Staubli VAL3: modIMM.pjx

--- modIMM.pjx ---
Parameters version=s7.2 stackSize=5000 millimeterUnit=true
Program file=_StartMachine.pgx
Program file=_WaitAuto.pgx
Program file=_WaitEnd.pgx
Program file=_WaitPart.pgx
Program file=_WaitPartDyn.pgx
Program file=BtRobotOff.pgx
Program file=checkMotStack.pgx
Program file=childAction.pgx
Program file=getSetting.pgx
Program file=IMMTiming.pgx
Program file=init.pgx
Program file=loadLibraries.pgx
Program file=primeAreaTest.pgx
Program file=primeMotStack.pgx
Program file=registerSetting.pgx
Program file=retrieveViews.pgx
Program file=runHigh.pgx
Program file=runLow.pgx
Program file=secuTask1.pgx
Program file=secuTask2.pgx
Program file=setDryRunSig.pgx
Program file=setSetting.pgx
Program file=slot.pgx
Program file=start.pgx
Program file=startAreaTest.pgx
Program file=stop.pgx
Program file=stopAreaTest.pgx
Program file=taskPartMade.pgx
Program file=updateView.pgx
Program file=WaitPart.pgx
Data file=modIMM.dtx
Library alias=io path=Disk://io/io.pjx
Library alias=SYS path=Disk://io_System/io_System.pjx
Library alias=scr path=Disk://Plastic/coreModules/modScreen/modScreen.pjx
Library alias=str path=Disk://Libraries/stringHandling/stringHandling.pjx
Library alias=lang path=Disk://Plastic/i18n/i18n.pjx
Library alias=debug path=Disk://Libraries/debug/debug.pjx
Library alias=data path=Disk://zData/zData.pjx
Library alias=status path=Disk://Plastic/coreModules/modStatusModel/modStatusModel.pjx
Library alias=EV path=Disk://Plastic/Consts/EVENT/EVENT.pjx
Library alias=sig path=Disk://Plastic/coreModules/modSignalSlot/modSignalSlot.pjx
Library alias=STATE path=Disk://Plastic/Consts/STATE/STATE.pjx
Library alias=views path=Disk://Plastic/coreModules/viewContainer/viewContainer.pjx
Library alias=jt path=Disk://Libraries/jointFunctions/jointFunctions.pjx
Type name=event path=Disk://Plastic/Types/event/event.pjx
Type name=settingType path=Disk://Plastic/Types/setting/setting.pjx
Type name=viewType path=Disk://Plastic/Types/view/view.pjx
Type name=childNodeType path=Disk://Plastic/Types/childNode/childNode.pjx
Type name=nodeType path=Disk://Plastic/Types/node/node.pjx

--- modIMM.dtx ---
num nCaseBtRobOff
num nStateRstPart[4]
num nStatePartMade
num reactionTime
num pointer
num timings[40]
public num nCloseDelayTime
num mouldTimer
bool bRobotOffAllow
bool bState
num tmMotionStack
num WAR_MOTIONSTACK = 1
bool bDisplayed
bool bSuspendForTest
num WAIT_MOULD_FREE
num nAreaTestState
num nMouldAreaZone
num WAIT_MOULD_OPEN
num WAIT_ROB_ENABLE
num WAIT_IMM_AUTO
num WAIT_PARTMADE
public string name = "IMM"
num moduleIndex
bool bAtWaitPosition
string IMM_IO_PTH
num nImmType
bool bRobotOff
num AREA_TEST_FAIL
num nMouldAreaDist
num HOME_IN_MOULD
num ARM_IN_MOULD_NO
num ARM_IN_MOULD_ST

--- start.pgx ---
public program start()
begin
  // set nCaseBtRobOff to 1 instead of 0 in order to initialize the robot off function properly
  // If nCaseBtRobOff is 0 at start up it may happen that SYS:doRobotOff["+toString("",moduleIndex)+"] is on although btRobotOff assumes that
  // SYS:doRobotOff["+toString("",moduleIndex)+"] is off.

  call debug:setVerbosity(libPath(),debug:LEV_INFO)
  call loadLibraries()
  // call setDryRunSig(data:setDryRun)
  call sig:connect(EV:DRY_RUN,libPath())
  call sig:connect(EV:FATAL_ERROR,libPath())
  call sig:connect(EV:START_COMPLETE,libPath())
  call status:registerStatus(libPath(),status:CL_STATUS,"Wait for mould free condition","SYS:doMouldFree["+toString("",moduleIndex)+"]==true","SYS:doMouldFree["+toString("",moduleIndex)+"]==false",false,WAIT_MOULD_FREE,false)
  call status:registerStatus(libPath(),status:CL_STATUS,"Wait for mould open","SYS:diMouldOpen["+toString("",moduleIndex)+"]==true","SYS:diMouldOpen["+toString("",moduleIndex)+"]==false",false,WAIT_MOULD_OPEN,false)
  call status:registerStatus(libPath(),status:CL_STATUS,"Wait for robot enabled","SYS:doRobotOff["+toString("",moduleIndex)+"]==false","SYS:doRobotOff["+toString("",moduleIndex)+"]==true",false,WAIT_ROB_ENABLE,false)
  call status:registerStatus(libPath(),status:CL_STATUS,"Wait for IMM in auto mode","SYS:diMachineInAuto["+toString("",moduleIndex)+"]==true","SYS:diMachineInAuto["+toString("",moduleIndex)+"]==false",false,WAIT_ROB_ENABLE,false)
  call status:registerStatus(libPath(),status:CL_STATUS,"Wait for part produced","SYS:bPartMade["+toString("",moduleIndex)+"]==true","SYS:bPartMade["+toString("",moduleIndex)+"]==false",false,WAIT_PARTMADE,false)
  call status:registerStatus(libPath(),status:CL_ERROR,"Mould area test failed. Robot was not programmed to enter mould","","",true,AREA_TEST_FAIL,true)
  call status:registerStatus(libPath(),status:CL_ERROR,"Home position is defined in mould area","","",true,HOME_IN_MOULD,true)
  call status:registerStatus(libPath(),status:CL_ERROR,"Arm in mould while mould is not open","","",true,ARM_IN_MOULD_NO,true)
  call status:registerStatus(libPath(),status:CL_ERROR,"Arm in mould while 'Enable Closure' signal is set","","",true,ARM_IN_MOULD_ST,true)
end

--- _StartMachine.pgx ---
public program _StartMachine()
// Start machine cycle
  local bool bAreaTest
  local num nOldSpeedScale
  local bool bTestRun
  local string txt
  local num time
  local string sValue
begin
  //
  // add list of pending status messages
  //!i18n 16 -> "Wait for Mould Free Condition"

  call status:setEnabled(WAIT_MOULD_FREE,true)
  //!change 23.05.06, vdg: reduce speed in test mode when approaching the mould area boundary
  // from inside towards outside
  //!change 08.09.06, vdg: store data:setTestRun in a local variable
  bTestRun=data:setTestRun
  // prime the motion stack monitor which checks if the arm is actually
  // programmed to leave the mould when StartMachine() is called
  call primeMotStack()
  if bTestRun
    //wait(secu:nSafeZoneDist[0]<300)
    nOldSpeedScale=getMonitorSpeed()
    //!fix 09.06.06, vdg: set speed to the lower speed setting (current speedScale() or dry run speed)
    ///TODO
    //$setSpeed(min(speedScale(),10))
    //call setSpeed(min(getMonitorSpeed(),10))
    //wait(secu:nSafeZoneDist[0]<50)
    //$setSpeed(1)
    ///TODO
    //call setSpeed(1)
  endIf
  // WAIT GRIPPER OUT OF MOULD AREA ==================================================================================
  // record the safety distance of the robot

  time=clock()
  //requiredTime=0.2
  //currentTime=0
  // if (speedScale()>99) and (workingMode()==4) and (SYS:diMachineInAuto[moduleIndex]==true) and !bTestRun
  if (getMonitorSpeed()>99) and (workingMode()==4) and !bTestRun
    do
      // Check if there are still motions in the stack.
      // If it is empty, it means the robot never leaves the mould area before
      // StartMachine() is called.
      call checkMotStack()
    until (SYS:doMouldFree[moduleIndex]==true)
  else
    do
      // Check if there are still motions in the stack.
      // If it is empty, it means the robot never leaves the mould area before
      // StartMachine() is called.
      call checkMotStack()
    until (SYS:doMouldFree[moduleIndex]==true)
  endIf
  //
  call status:setEnabled(WAIT_MOULD_FREE,false)
  //
  //!change 18.05.06, vdg: check if doMouldFree has toggled
  call stopAreaTest(bAreaTest)
  // START MACHINE CYCLE =============================================================================================
  //!change 16.02.06, vdg: Allow to start IMM in endIf cycle mode SYS:bStartInEndCycl is set
  if (!SYS:CE_Requested or SYS:bStartInEndCycl) and !SYS:bPartMade[moduleIndex] and bAreaTest
    //!change 18.05.06, vdg: Stop robot at point where machine is being started
    //  and ask the user if it is safe to start the IMM
    if bTestRun
      bSuspendForTest=true
      // reset original speedScale only if speed was not modified by user meanwhile
      // wait for settled arm
      watch(isSettled(),3)
      // reset old speed setting if it wasn't changed by the user
      if getMonitorSpeed()==1
        ///TODO
        //$setSpeed(nOldSpeedScale)
        //call setSpeed(nOldSpeedScale)
      endIf
      //sValue=toString("4.0",secu:nSafeZoneDist[0])
      call str:printf((("Robot stopped approx. at point where IMM cycle is being started (Overshoot: %1mm). Press START to continue!")),sValue,txt)
      ///TODO
      //call ui:popUpCond(txt,"SYS:bBtStart==true",false)
      bSuspendForTest=true
      wait(bSuspendForTest==false)
    endIf
    //!change 08.06.06, vdg: Start IMM only if dry run mode is not active
    if !bTestRun
      SYS:doStartMachine[moduleIndex]=true
    endIf
    //call stat:stopTakeTime()
    //call stat:stopCycleTime()
    //call stat:startCycleTime()
    //call stat:startRobotTime()
  endIf
  //
end

--- _WaitPartDyn.pgx ---
public program _WaitPartDyn()
// Wait part made in machine and mould fully open
begin
  //!brief
  // Wait for a part being made and conditions for the robot to enter mold.
  //
  call WaitPart(true)
end

--- checkMotStack.pgx ---
program checkMotStack()
begin
  //!brief
  //This routine sets a warnig if the motion stack has been empty for more than WAR_MOTIONSTACK seconds.

  if (clock()-tmMotionStack>WAR_MOTIONSTACK) and !bDisplayed and isEmpty()
    ///TODO
    //call status:raise()
    //call ui:popUp((("The routine StartMachine() was called, but the arm is not programmed to leave the mould!")),data:nMsgTimeOut,false)
    bDisplayed=true
  endIf
end

--- init.pgx ---
public program init()
  local bool ok
  local string path
  local num idx
begin
  // set module index
  path=libPath()
  path=right(path,1)
  path=toNum(path,moduleIndex,ok)
  if !ok
    moduleIndex=0
  endIf
  name="IMM"+toString("1.0",moduleIndex)
  IMM_IO_PTH="2:IO/1:"+name
  nCaseBtRobOff=1
  bState=false
  pointer=0
  for idx=0 to size(timings)-1
    timings[idx]=0
  endFor

end

--- retrieveViews.pgx ---
public program retrieveViews(viewType& view_, num& idx_)
begin
  switch idx_
    case 0
      view_.path=IMM_IO_PTH
      view_.label="IMM"
      call views:appendNode(view_.nodes,"Safety")
      call views:appendNode(view_.nodes,"Machine")
      call views:appendNode(view_.nodes,"Ejectors")
      call views:appendNode(view_.nodes,"Cores")
      call views:appendNode(view_.nodes,"Mould")
      view_.type=view_.TYPE_TREEVIEW
    break
  endSwitch
end

--- run.pgx ---
public program run()
begin
  call taskPartMade()
  call IMMTiming()
end

--- runLow.pgx ---
public program runLow()
begin
  if data:setDryRun==true
    if SYS:diMachineInAuto[moduleIndex]==true
      data:setDryRun=false
      call scr:popUp("Dry run mode automatically deactivated because IMM is in 'Automatic' mode!",data:nMsgTimeOut,false)
    endIf
    if bRobotOff==true
      data:setDryRun=false
      call scr:popUp("Dry run mode automatically deactivated because robot is disabled!",data:nMsgTimeOut,false)
    endIf
  endIf
end

--- secuTask2.pgx ---
public program secuTask2()
// Control of Safety realay
  local point pLocFlange
  local point pLocTCP
begin
  // wait until system is initialized
  if SYS:nStateRobot<=STATE:INITIALIZING
    return
  endIf
  if SYS:doSecu[0]==false or SYS:doSecu[1]==false
    return
  endIf
  // Get home position relative to the frame of IMM mould area.....
  if jt:isTXRobot
    pLocFlange=jointToPoint(flange,data:fAreaIMM,data:jHomeTX)
    pLocTCP=jointToPoint(data:tTCP,data:fAreaIMM,data:jHomeTX)
  else
    pLocFlange=jointToPoint(flange,data:fAreaIMM,data:jHomeTS)
    pLocTCP=jointToPoint(data:tTCP,data:fAreaIMM,data:jHomeTS)
  endIf
//
  if pLocTCP.trsf.z>nMouldAreaZone
    call status:raise(HOME_IN_MOULD,"")
  endIf
  // Get current robot position relative to the frame of IMM Backside.....
  pLocFlange=here(flange,data:fAreaIMM)
  pLocTCP=here(data:tTCP,data:fAreaIMM)
  nMouldAreaDist=max(pLocTCP.trsf.z,pLocFlange.trsf.z)-nMouldAreaZone
  //
  // Robotarm in mould when sig:MouldOpen missing or sig:StartIMM is active..........................................................
  if SYS:doMouldFree==false and (SYS:diMouldMidOpen==false and SYS:diMouldOpen==false)
    call status:raise(ARM_IN_MOULD_NO,"")
  endIf
  if (SYS:doMouldFree==false and SYS:doStartMachine==true)
    call status:raise(ARM_IN_MOULD_ST,"")
  endIf
end

--- setDryRunSig.pgx ---
public program setDryRunSig(bool enable_)
begin
  if enable_
    call debug:warning(libPath(),"Dry run mode enabled")
    dioLink(SYS:diEjcIn,SYS:doEjcIn)
    dioLink(SYS:diEjcOut,SYS:doEjcOut)
    dioLink(SYS:diCore1Pos1,SYS:doCore1Pos1)
    dioLink(SYS:diCore1Pos2,SYS:doCore1Pos2)
    dioLink(SYS:diCore2Pos1,SYS:doCore2Pos1)
    dioLink(SYS:diCore2Pos2,SYS:doCore2Pos2)
  else
    call debug:warning(libPath(),"Dry run mode disabled")
    call SYS:InitSysIO()
  endIf
end

--- setSetting.pgx ---
public program setSetting(settingType setting_)
begin
  switch setting_.sType
    case "num"
      $exec(setting_.varName+"=setting_.nValue")
    break
    case "bool"
      $exec(setting_.varName+"=setting_.bValue")
    break
    case "string"
      $exec(setting_.varName+"=setting_.sValue")
    break
  endSwitch
end

--- slot.pgx ---
public program slot(event& event_)
begin
  switch event_.nType
    case EV:DRY_RUN
      call setDryRunSig(event_.sParam=="1")
    break
    case EV:START_COMPLETE
      SYS:doSecu[0]=true
    SYS:doSecu[1]=true
    break
  endSwitch
end

--- stopAreaTest.pgx ---
public program stopAreaTest(bool& bResult_[])
begin
  // test result of area test state machine
  // the state nAreaTestState must be 40
  if nAreaTestState!=40 and nAreaTestState!=0
    call status:raise(AREA_TEST_FAIL,"")
  endIf
  bResult_=nAreaTestState==40 or nAreaTestState==0
end

--- updateView.pgx ---
public program updateView()
  local string sValues[5]
  local childNodeType child
begin

  call views:childDIO(views:views[IMM_IO_PTH].nodes[0],0,"Safety Relay 1",SYS:doSecu[0])
  call views:childDIO(views:views[IMM_IO_PTH].nodes[0],1,"Safety Relay 2",SYS:doSecu[1])

  sValues[0]=toString("4.0",nMouldAreaDist)
  if SYS:doMouldFree[moduleIndex]==true
    sValues[1]="/ti"
  endIf
  call str:printf(("%2 %1/tnmm"),sValues,child.valueText)
  child.label="Safety Distance"
  call views:setChild(views:views[IMM_IO_PTH].nodes[0],2,child)

  call views:childDIO(views:views[IMM_IO_PTH].nodes[1],0,"Robot Off",SYS:doRobotOff[moduleIndex])
  call views:childDIO(views:views[IMM_IO_PTH].nodes[1],1,"Mould Area Free",SYS:doMouldFree[moduleIndex])
  call views:childDIO(views:views[IMM_IO_PTH].nodes[1],2,"Enable Mould Closure",SYS:doStartMachine[moduleIndex])
  call views:childDIO(views:views[IMM_IO_PTH].nodes[1],3,"Automatic Mode",SYS:diMachineInAuto[moduleIndex])
  call views:childDIO(views:views[IMM_IO_PTH].nodes[1],4,"Reject Part",SYS:diRejectPart[moduleIndex])

  call views:childDIO(views:views[IMM_IO_PTH].nodes[2],0,"Ejector forward",SYS:doEjcOut[moduleIndex])
  call views:childDIO(views:views[IMM_IO_PTH].nodes[2],1," ",SYS:diEjcOut[moduleIndex])
  call views:childDIO(views:views[IMM_IO_PTH].nodes[2],2,"Ejector forward",SYS:doEjcIn[moduleIndex])
  call views:childDIO(views:views[IMM_IO_PTH].nodes[2],3," ",SYS:diEjcIn[moduleIndex])

  call views:childDIO(views:views[IMM_IO_PTH].nodes[3],0,"Core 1 Pos 1",SYS:doCore1Pos1[moduleIndex])
  call views:childDIO(views:views[IMM_IO_PTH].nodes[3],1," ",SYS:diCore1Pos1[moduleIndex])
  call views:childDIO(views:views[IMM_IO_PTH].nodes[3],2,"Core 1 Pos 2",SYS:doCore1Pos2[moduleIndex])
  call views:childDIO(views:views[IMM_IO_PTH].nodes[3],3," ",SYS:diCore1Pos2[moduleIndex])
  call views:childDIO(views:views[IMM_IO_PTH].nodes[3],4,"Core 2 Pos 1",SYS:doCore2Pos1[moduleIndex])
  call views:childDIO(views:views[IMM_IO_PTH].nodes[3],5," ",SYS:diCore1Pos1[moduleIndex])
  call views:childDIO(views:views[IMM_IO_PTH].nodes[3],6,"Core 2 Pos 2",SYS:doCore2Pos2[moduleIndex])
  call views:childDIO(views:views[IMM_IO_PTH].nodes[3],7," ",SYS:diCore1Pos2[moduleIndex])


  call views:childDIO(views:views[IMM_IO_PTH].nodes[4],0,"Mould Open",SYS:doFullOpening[moduleIndex])
  call views:childDIO(views:views[IMM_IO_PTH].nodes[4],1," ",SYS:diMouldOpen[moduleIndex])
  call views:childDIO(views:views[IMM_IO_PTH].nodes[4],2,"Mould Closed",SYS:diMouldClosed[moduleIndex])
  call views:childDIO(views:views[IMM_IO_PTH].nodes[4],3,"Mould Intermediate Pos",SYS:diMouldMidOpen[moduleIndex])
end
